FUNCTION CADD : complex
VAR_INPUT
	X, Y : complex;
END_VAR


(*
version 1.0	21 feb 2008
programmer 	hugo
tested by	oscat

this function add two complex numbers

*)

CADD.re := x.re + y.re;
CADD.im := x.im + y.im;


(* revision history
hm	21. feb 2008	rev 1.0
	original version

*)

END_FUNCTION

(* stored: Version 1.1.0.1, ProductVersion 3.1.4022.7
   POU CADD: Id {ca736068-9c3e-430c-b1fb-cdf866061e82}, SpecialFunc None *)
